Yaskawa INFORM job: _DEL196.JBI

/JOB
//NAME _DEL196
//POS
///NPOS 0,0,0,0,0,1
///TOOL 0
///POSTYPE ANGLE
///ANGLE
EX00110=0.0000
//INST
///DATE 2018/11/14 13:43
///ATTR SC,RW,SY
///GROUP1 ST1
///LVARS 5,0,5,0,0,0,0,0
NOP
*top
GETS PX110 $PX001
GETE LD000 EX110 (1)
DIV LD000 20000
IFTHEN LD000>1
	 SET LB000 LD000
	 DOUT OG#(82) LB000
ENDIF
DELAY 200
JUMP *top
END
